// TIA Portal project "phanloai_demo" (V16)

(* hardware
DEVICE "S7-1200 station_1"  S7-1200 Station
   slot 0: "Rack_0"  S7-1200 Rack  Rack  V1.0
   slot 1: "PLC_1"  CPU 1214C DC/DC/DC  6ES7 214-1AG40-0XB0  V4.4
*)

// ===== PLC "PLC_1"  CPU 1214C DC/DC/DC =====

VAR_GLOBAL   // PLC tag table "Default tag table"
   "pulse_I0.7" AT %M50.0 : Bool;
   "pulse_nanglen1" AT %M50.4 : Bool;
   "pulse_haxuong" AT %M50.5 : Bool;
   "pulse_nanglen2" AT %M50.6 : Bool;
   "pulse_haxuong1" AT %M51.0 : Bool;
   "pulse_dira" AT %M51.2 : Bool;
   "pulse_covat" AT %M61.2 : Bool;
   "pulse_vatcuoi" AT %M62.3 : Bool;
   "pulse_run" AT %M62.4 : Bool;
   "pulse_MQTT_VT2" AT %M70.1 : Bool;
   "pulse_MQTT_VT1" AT %M70.0 : Bool;
   "pulse_MQTT_VT3" AT %M70.2 : Bool;
   "pulse_VT1" AT %M63.0 : Bool;
   "pulse_dive" AT %M62.5 : Bool;
   "Tag_3" AT %M51.4 : Bool;
   "pulse_VT2" AT %M63.1 : Bool;
   "pulse_VT3" AT %M63.2 : Bool;
   "pulse_nanglen_2" AT %M62.6 : Bool;
   "Tag_5" AT %M62.7 : Bool;
   "pulse_emer" AT %M9.3 : Bool;
   "Tag_4" AT %M9.4 : Bool;
   "Tag_6" AT %M15.0 : Bool;
   "Tag_7" AT %M15.1 : Bool;
   "Tag_8" AT %M15.2 : Bool;
   "undefine" AT %M2.5 : Bool;
   "Tag_9" AT %M2.6 : Bool;
   "Tag_10" AT %M2.7 : Bool;
   "ready" AT %M4.7 : Bool;
   "not_ready" AT %M4.6 : Bool;
   "Tag_11" AT %M5.5 : Bool;
   "Tag_12" AT %M5.6 : Bool;
   "Tag_13" AT %M5.7 : Bool;
   "stop_QR" AT %M9.5 : Bool;
   "QR_check" AT %M9.6 : Bool;
   "mode" AT %M9.7 : Bool;
   "Color_check" AT %M12.5 : Bool;
END_VAR

VAR_GLOBAL   // PLC tag table "Input"
   "Button_start" AT %I0.0 : Bool;
   "CB_covat" AT %I0.1 : Bool;
   "CB_dua_vat_ve" AT %I0.2 : Bool;
   "CB_day_vat_ra" AT %I0.3 : Bool;
   "CB_dira_2" AT %I0.4 : Bool;
   "CB_vatcuoi" AT %I0.7 : Bool;
   "CB_dive" AT %I1.0 : Bool;
   "CB_dira_1" AT %I1.1 : Bool;
   "CB_dira_3" AT %I1.2 : Bool;
   "CB_nanglen" AT %I1.3 : Bool;
   "CB_haxuong" AT %I1.4 : Bool;
   "Button_reset" AT %I1.5 : Bool;
END_VAR

VAR_GLOBAL   // PLC tag table "Output"
   "motor" AT %Q0.0 : Bool;
   "kep_phoi" AT %Q0.1 : Bool;
   "nanglen" AT %Q0.2 : Bool;
   "dive" AT %Q0.3 : Bool;
   "day_vat_ra" AT %Q0.4 : Bool;
   "nha_phoi" AT %Q0.5 : Bool;
   "haxuong" AT %Q0.6 : Bool;
   "dira" AT %Q0.7 : Bool;
   "dua_vat_ve" AT %Q1.1 : Bool;
END_VAR

VAR_GLOBAL   // PLC tag table "Memory"
   "Tag_1" AT %M0.0 : Bool;
   "Tag_2" AT %M0.1 : Bool;
   "reset_run" AT %M1.0 : Bool;
   "M_day_vat_ve" AT %M1.1 : Bool;
   "M_day_vat_ra" AT %M1.4 : Bool;
   "ha_xuong_1" AT %M2.0 : Bool;
   "nang_len_1" AT %M2.1 : Bool;
   "ha_xuong_2" AT %M2.2 : Bool;
   "nang_len_2" AT %M2.3 : Bool;
   "M_dive" AT %M2.4 : Bool;
   "dua_vat_ve_reset" AT %M3.0 : Bool;
   "nang_len_reset" AT %M3.1 : Bool;
   "dive_reset" AT %M3.2 : Bool;
   "nha_phoi_reset" AT %M3.3 : Bool;
   "co_vat" AT %M3.4 : Bool;
   "Run" AT %M3.5 : Bool;
   "motor_on" AT %M10.0 : Bool;
   "dayvat_ra_on" AT %M10.1 : Bool;
   "duavat_ve_on" AT %M10.2 : Bool;
   "dive_on" AT %M10.3 : Bool;
   "dira_on" AT %M10.4 : Bool;
   "nanglen_on" AT %M10.5 : Bool;
   "haxuong_on" AT %M10.6 : Bool;
   "kep_phoi_on" AT %M10.7 : Bool;
   "nha_phoi_on" AT %M11.0 : Bool;
   "SP1" AT %M12.0 : Bool;
   "dira_stop" AT %M12.1 : Bool;
   "VT1" AT %M12.2 : Bool;
   "VT2" AT %M12.3 : Bool;
   "VT3" AT %M12.4 : Bool;
   "M_stop" AT %M1.2 : Bool;
   "SL_VT1" AT %MW150 : UInt;
   "SL_VT2" AT %MW152 : UInt;
   "SL_VT3" AT %MW154 : UInt;
   "off_nha_phoi" AT %M3.6 : Bool;
   "off_nang_len" AT %M3.7 : Bool;
   "Auto_mode" AT %M1.3 : Bool;
   "Man_mode" AT %M1.7 : Bool;
   "Auto_run" AT %M4.0 : Bool;
   "Man_run" AT %M4.1 : Bool;
   "reset_VT1" AT %M4.2 : Bool;
   "reset_VT2" AT %M4.3 : Bool;
   "reset_VT3" AT %M4.4 : Bool;
   "stop_reset" AT %M4.5 : Bool;
   "Emer_on" AT %M5.0 : Bool;
   "Emer_run" AT %M5.2 : Bool;
   "Emer_off" AT %M5.1 : Bool;
   "S1" AT %M8.0 : Bool;
   "S2" AT %M8.1 : Bool;
   "S3" AT %M8.2 : Bool;
   "S5" AT %M8.4 : Bool;
   "S4" AT %M8.3 : Bool;
   "S6" AT %M8.5 : Bool;
   "S10" AT %M9.1 : Bool;
   "S9" AT %M9.0 : Bool;
   "S8" AT %M8.7 : Bool;
   "S7" AT %M8.6 : Bool;
END_VAR

DATA_BLOCK "Receive data MQTT"   // DB1
{ S7_Optimized_Access := 'FALSE' }
VERSION : 0.1
   VAR
      VT1 : Bool;
      VT2 : Bool;
      VT3 : Bool;
      Start : Bool;
      Stop : Bool;
      Reset : Bool;
      Emergency : Bool;
      Man_day_vat_ra : Bool;
      Man_dua_vat_ve : Bool;
      Man_haxuong : Bool;
      Man_nanglen : Bool;
      Man_kepphoi : Bool;
      Man_nhaphoi : Bool;
      Man_dira : Bool;
      Man_dive : Bool;
      Man_bangtai : Bool;
   END_VAR
BEGIN
END_DATA_BLOCK

DATA_BLOCK "Send data MQTT"   // DB2
{ S7_Optimized_Access := 'FALSE' }
VERSION : 0.1
   VAR
      SL_VT1 : Int;
      SL_VT2 : Int;
      SL_VT3 : Int;
   END_VAR
BEGIN
END_DATA_BLOCK

DATA_BLOCK "Manual"   // DB4
{ S7_Optimized_Access := 'FALSE' }
VERSION : 0.1
   VAR
      Man_motor_on : Bool;
      Man_motor_off : Bool;
      Man_dua_vat_ve : Bool;
      Man_day_vat_ra : Bool;
      Man_haxuong : Bool;
      Man_nanglen : Bool;
      Man_kepphoi : Bool;
      Man_nhaphoi : Bool;
      Man_dira : Bool;
      Man_dive : Bool;
   END_VAR
BEGIN
END_DATA_BLOCK

// folder: System blocks/Program resources

DATA_BLOCK "QR_delay"   // DB3
{ S7_Optimized_Access := 'TRUE' }
AUTHOR : Simatic
FAMILY : IEC
NAME : IEC_TMR
VERSION : 1.0
// stored: InstanceOfName IEC_TIMER
"IEC_TIMER"
BEGIN
END_DATA_BLOCK

DATA_BLOCK "QR_stop"   // DB5
{ S7_Optimized_Access := 'TRUE' }
AUTHOR : Simatic
FAMILY : IEC
NAME : IEC_TMR
VERSION : 1.0
// stored: InstanceOfName IEC_TIMER
"IEC_TIMER"
BEGIN
END_DATA_BLOCK

// folder: (top level)

FUNCTION "Auto" : Void   // FC1, LAD
{ S7_Optimized_Access := 'TRUE' }
VERSION : 0.1
   VAR_INPUT
      Button_start : Bool;
      CB_covat : Bool;
      CB_dua_vat_ve : Bool;
      CB_day_vat_ra : Bool;
      CB_dira_2 : Bool;
      CB_vatcuoi : Bool;
      CB_dive : Bool;
      CB_dira_1 : Bool;
      CB_dira_3 : Bool;
      CB_nanglen : Bool;
      CB_haxuong : Bool;
      MQTT_VT1 : Bool;
      MQTT_VT2 : Bool;
      MQTT_VT3 : Bool;
      MQTT_start : Bool;
      MQTT_stop : Bool;
      MQTT_emer : Bool;
      reset_run : Bool;
      Emer_on : Bool;
      Emer_run : Bool;
   END_VAR
   VAR_OUTPUT
      motor : Bool;
      nanglen : Bool;
      haxuong : Bool;
   END_VAR
   VAR_IN_OUT
      SL_VT1 : Int;
      SL_VT2 : Int;
      SL_VT3 : Int;
      day_vat_ra : Bool;
      dua_vat_ve : Bool;
      kep_phoi : Bool;
      dira : Bool;
      nha_phoi : Bool;
      dive : Bool;
   END_VAR
   VAR_TEMP   // added for the SCL form of the ladder/FBD networks
      _w1 : Bool;
      _w2 : Bool;
      _w3 : Bool;
      _w4 : Bool;
      _w5 : Bool;
   END_VAR
BEGIN

REGION Network 1
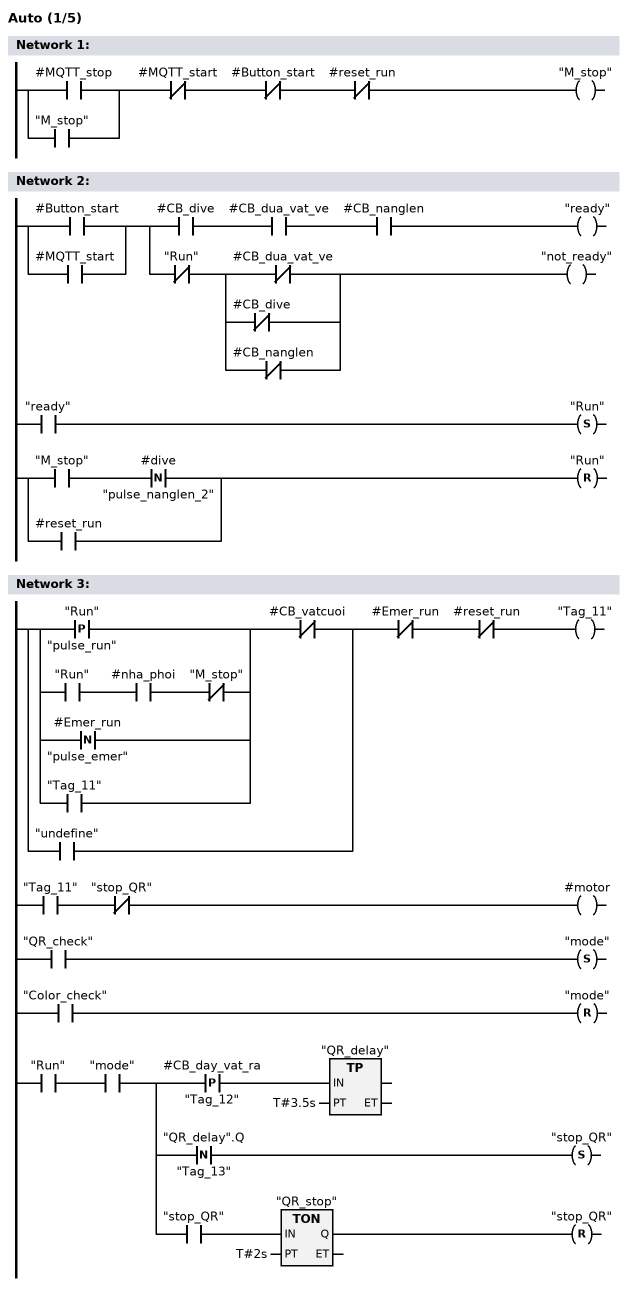
   RUNG wire#powerrail
      Contact( #MQTT_stop )
      wire#w1
      I_Contact( #MQTT_start )
      I_Contact( #Button_start )
      I_Contact( #reset_run )
      Coil( "M_stop" )
   END_RUNG
   RUNG wire#powerrail
      Contact( "M_stop" )
   END_RUNG wire#w1
   // the same network as SCL:
   "M_stop" := (#MQTT_stop OR "M_stop") AND NOT #MQTT_start AND NOT #Button_start AND NOT #reset_run;
END_REGION

REGION Network 2
   RUNG wire#powerrail
      Contact( #Button_start )
      wire#w1
      Contact( #CB_dive )
      Contact( #CB_dua_vat_ve )
      Contact( #CB_nanglen )
      Coil( "ready" )
   END_RUNG
   RUNG wire#powerrail
      Contact( #MQTT_start )
   END_RUNG wire#w1
   RUNG wire#w1
      I_Contact( "Run" )
      wire#w2
      I_Contact( #CB_dua_vat_ve )
      wire#w3
      Coil( "not_ready" )
   END_RUNG
   RUNG wire#w2
      I_Contact( #CB_dive )
   END_RUNG wire#w3
   RUNG wire#w2
      I_Contact( #CB_nanglen )
   END_RUNG wire#w3
   RUNG wire#powerrail
      Contact( "ready" )
      S_Coil( "Run" )
   END_RUNG
   RUNG wire#powerrail
      Contact( "M_stop" )
      N_Contact(operand := #dive, bit := "pulse_nanglen_2")
      wire#w4
      R_Coil( "Run" )
   END_RUNG
   RUNG wire#powerrail
      Contact( #reset_run )
   END_RUNG wire#w4
   // the same network as SCL:
   #_w1 := #Button_start OR #MQTT_start;
   "ready" := #_w1 AND #CB_dive AND #CB_dua_vat_ve AND #CB_nanglen;
   "not_ready" := #_w1 AND NOT "Run" AND (NOT #CB_dua_vat_ve OR NOT #CB_dive OR NOT #CB_nanglen);
   IF "ready" THEN "Run" := TRUE; END_IF;
   #_w2 := "M_stop" AND NOT #dive AND "pulse_nanglen_2";   // falling edge of #dive
   "pulse_nanglen_2" := #dive;
   IF #_w2 OR #reset_run THEN "Run" := FALSE; END_IF;
END_REGION

REGION Network 3
   #_w1 := "Run" AND NOT "pulse_run";   // rising edge of "Run"
   "pulse_run" := "Run";
   #_w2 := NOT #Emer_run AND "pulse_emer";   // falling edge of #Emer_run
   "pulse_emer" := #Emer_run;
   "Tag_11" := (((#_w1 OR ("Run" AND #nha_phoi AND NOT "M_stop") OR #_w2 OR "Tag_11") AND NOT #CB_vatcuoi) OR "undefine") AND NOT #Emer_run AND NOT #reset_run;
   #motor := "Tag_11" AND NOT "stop_QR";
   IF "QR_check" THEN "mode" := TRUE; END_IF;
   IF "Color_check" THEN "mode" := FALSE; END_IF;
   #_w3 := "Run" AND "mode";
   #_w4 := #_w3 AND #CB_day_vat_ra AND NOT "Tag_12";   // rising edge of #CB_day_vat_ra
   "Tag_12" := #CB_day_vat_ra;
   "QR_delay".TP(IN := #_w4, PT := T#3.5s);
   #_w5 := #_w3 AND NOT "QR_delay".Q AND "Tag_13";   // falling edge of "QR_delay".Q
   "Tag_13" := "QR_delay".Q;
   IF #_w5 THEN "stop_QR" := TRUE; END_IF;
   "QR_stop".TON(IN := #_w3 AND "stop_QR", PT := T#2s);
   IF "QR_stop".Q THEN "stop_QR" := FALSE; END_IF;
END_REGION

REGION Network 4
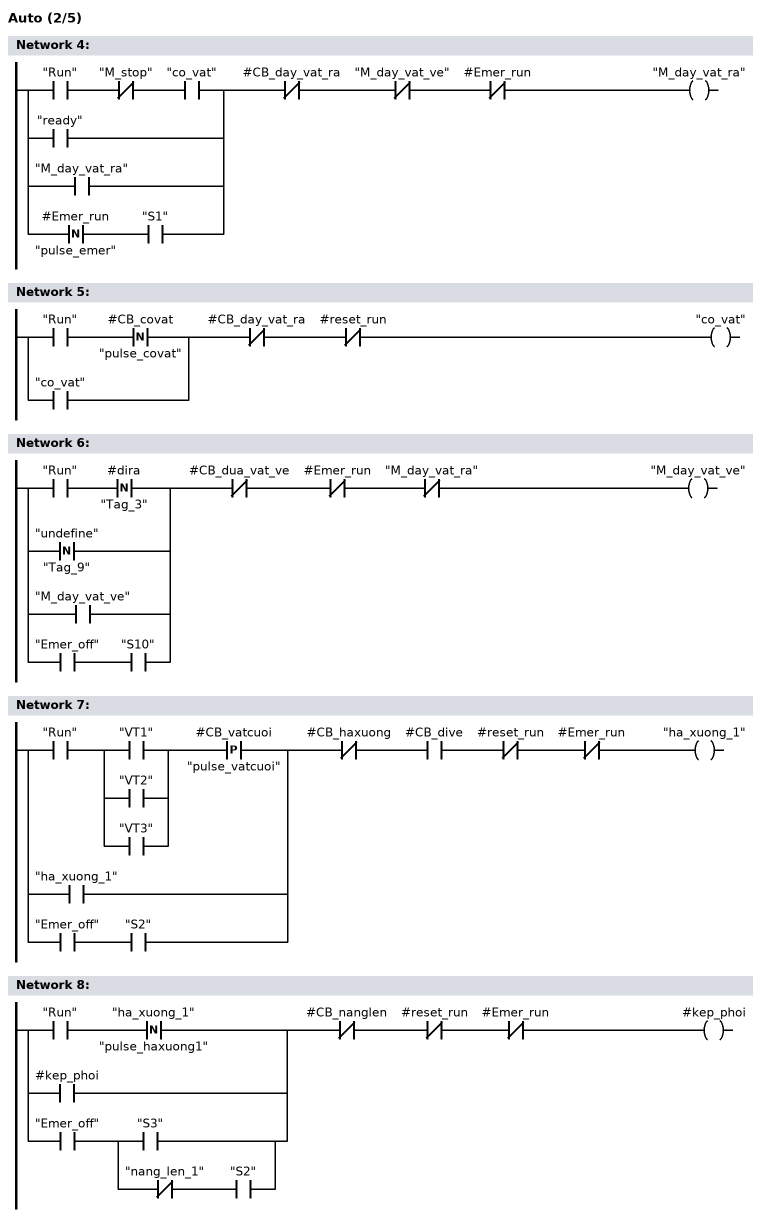
   RUNG wire#powerrail
      Contact( "Run" )
      I_Contact( "M_stop" )
      Contact( "co_vat" )
      wire#w1
      I_Contact( #CB_day_vat_ra )
      I_Contact( "M_day_vat_ve" )
      I_Contact( #Emer_run )
      Coil( "M_day_vat_ra" )
   END_RUNG
   RUNG wire#powerrail
      Contact( "ready" )
   END_RUNG wire#w1
   RUNG wire#powerrail
      Contact( "M_day_vat_ra" )
   END_RUNG wire#w1
   RUNG wire#powerrail
      N_Contact(operand := #Emer_run, bit := "pulse_emer")
      Contact( "S1" )
   END_RUNG wire#w1
   // the same network as SCL:
   #_w1 := NOT #Emer_run AND "pulse_emer";   // falling edge of #Emer_run
   "pulse_emer" := #Emer_run;
   "M_day_vat_ra" := (("Run" AND NOT "M_stop" AND "co_vat") OR "ready" OR "M_day_vat_ra" OR (#_w1 AND "S1")) AND NOT #CB_day_vat_ra AND NOT "M_day_vat_ve" AND NOT #Emer_run;
END_REGION

REGION Network 5
   RUNG wire#powerrail
      Contact( "Run" )
      N_Contact(operand := #CB_covat, bit := "pulse_covat")
      wire#w1
      I_Contact( #CB_day_vat_ra )
      I_Contact( #reset_run )
      Coil( "co_vat" )
   END_RUNG
   RUNG wire#powerrail
      Contact( "co_vat" )
   END_RUNG wire#w1
   // the same network as SCL:
   #_w1 := "Run" AND NOT #CB_covat AND "pulse_covat";   // falling edge of #CB_covat
   "pulse_covat" := #CB_covat;
   "co_vat" := (#_w1 OR "co_vat") AND NOT #CB_day_vat_ra AND NOT #reset_run;
END_REGION

REGION Network 6
   RUNG wire#powerrail
      Contact( "Run" )
      N_Contact(operand := #dira, bit := "Tag_3")
      wire#w1
      I_Contact( #CB_dua_vat_ve )
      I_Contact( #Emer_run )
      I_Contact( "M_day_vat_ra" )
      Coil( "M_day_vat_ve" )
   END_RUNG
   RUNG wire#powerrail
      N_Contact(operand := "undefine", bit := "Tag_9")
   END_RUNG wire#w1
   RUNG wire#powerrail
      Contact( "M_day_vat_ve" )
   END_RUNG wire#w1
   RUNG wire#powerrail
      Contact( "Emer_off" )
      Contact( "S10" )
   END_RUNG wire#w1
   // the same network as SCL:
   #_w1 := "Run" AND NOT #dira AND "Tag_3";   // falling edge of #dira
   "Tag_3" := #dira;
   #_w2 := NOT "undefine" AND "Tag_9";   // falling edge of "undefine"
   "Tag_9" := "undefine";
   "M_day_vat_ve" := (#_w1 OR #_w2 OR "M_day_vat_ve" OR ("Emer_off" AND "S10")) AND NOT #CB_dua_vat_ve AND NOT #Emer_run AND NOT "M_day_vat_ra";
END_REGION

REGION Network 7
   RUNG wire#powerrail
      Contact( "Run" )
      wire#w1
      Contact( "VT1" )
      wire#w2
      P_Contact(operand := #CB_vatcuoi, bit := "pulse_vatcuoi")
      wire#w3
      I_Contact( #CB_haxuong )
      Contact( #CB_dive )
      I_Contact( #reset_run )
      I_Contact( #Emer_run )
      Coil( "ha_xuong_1" )
   END_RUNG
   RUNG wire#w1
      Contact( "VT2" )
   END_RUNG wire#w2
   RUNG wire#w1
      Contact( "VT3" )
   END_RUNG wire#w2
   RUNG wire#powerrail
      Contact( "ha_xuong_1" )
   END_RUNG wire#w3
   RUNG wire#powerrail
      Contact( "Emer_off" )
      Contact( "S2" )
   END_RUNG wire#w3
   // the same network as SCL:
   #_w1 := "Run" AND ("VT1" OR "VT2" OR "VT3") AND #CB_vatcuoi AND NOT "pulse_vatcuoi";   // rising edge of #CB_vatcuoi
   "pulse_vatcuoi" := #CB_vatcuoi;
   "ha_xuong_1" := (#_w1 OR "ha_xuong_1" OR ("Emer_off" AND "S2")) AND NOT #CB_haxuong AND #CB_dive AND NOT #reset_run AND NOT #Emer_run;
END_REGION

REGION Network 8
   RUNG wire#powerrail
      Contact( "Run" )
      N_Contact(operand := "ha_xuong_1", bit := "pulse_haxuong1")
      wire#w1
      I_Contact( #CB_nanglen )
      I_Contact( #reset_run )
      I_Contact( #Emer_run )
      Coil( #kep_phoi )
   END_RUNG
   RUNG wire#powerrail
      Contact( #kep_phoi )
   END_RUNG wire#w1
   RUNG wire#powerrail
      Contact( "Emer_off" )
      wire#w2
      Contact( "S3" )
   END_RUNG wire#w1
   RUNG wire#w2
      I_Contact( "nang_len_1" )
      Contact( "S2" )
   END_RUNG wire#w1
   // the same network as SCL:
   #_w1 := "Run" AND NOT "ha_xuong_1" AND "pulse_haxuong1";   // falling edge of "ha_xuong_1"
   "pulse_haxuong1" := "ha_xuong_1";
   #kep_phoi := (#_w1 OR #kep_phoi OR ("Emer_off" AND ("S3" OR (NOT "nang_len_1" AND "S2")))) AND NOT #CB_nanglen AND NOT #reset_run AND NOT #Emer_run;
END_REGION

REGION Network 9
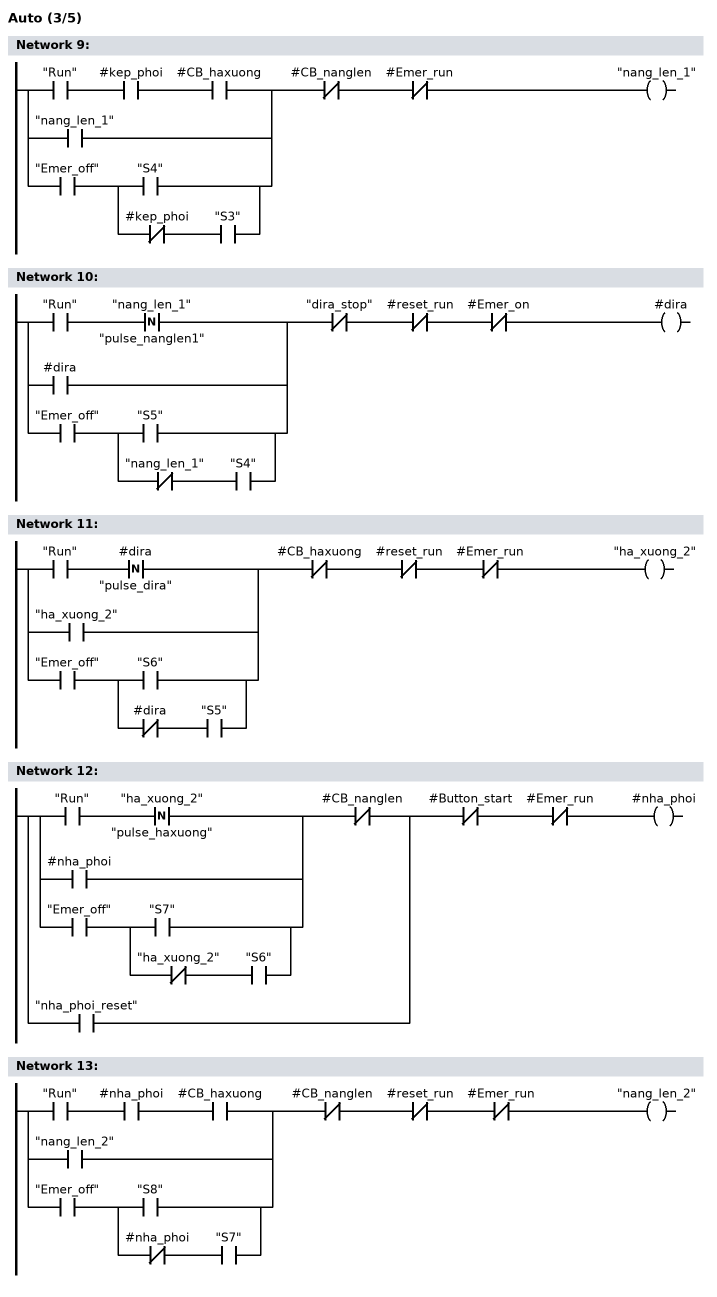
   RUNG wire#powerrail
      Contact( "Run" )
      Contact( #kep_phoi )
      Contact( #CB_haxuong )
      wire#w1
      I_Contact( #CB_nanglen )
      I_Contact( #Emer_run )
      Coil( "nang_len_1" )
   END_RUNG
   RUNG wire#powerrail
      Contact( "nang_len_1" )
   END_RUNG wire#w1
   RUNG wire#powerrail
      Contact( "Emer_off" )
      wire#w2
      Contact( "S4" )
   END_RUNG wire#w1
   RUNG wire#w2
      I_Contact( #kep_phoi )
      Contact( "S3" )
   END_RUNG wire#w1
   // the same network as SCL:
   "nang_len_1" := (("Run" AND #kep_phoi AND #CB_haxuong) OR "nang_len_1" OR ("Emer_off" AND ("S4" OR (NOT #kep_phoi AND "S3")))) AND NOT #CB_nanglen AND NOT #Emer_run;
END_REGION

REGION Network 10
   RUNG wire#powerrail
      Contact( "Run" )
      N_Contact(operand := "nang_len_1", bit := "pulse_nanglen1")
      wire#w1
      I_Contact( "dira_stop" )
      I_Contact( #reset_run )
      I_Contact( #Emer_on )
      Coil( #dira )
   END_RUNG
   RUNG wire#powerrail
      Contact( #dira )
   END_RUNG wire#w1
   RUNG wire#powerrail
      Contact( "Emer_off" )
      wire#w2
      Contact( "S5" )
   END_RUNG wire#w1
   RUNG wire#w2
      I_Contact( "nang_len_1" )
      Contact( "S4" )
   END_RUNG wire#w1
   // the same network as SCL:
   #_w1 := "Run" AND NOT "nang_len_1" AND "pulse_nanglen1";   // falling edge of "nang_len_1"
   "pulse_nanglen1" := "nang_len_1";
   #dira := (#_w1 OR #dira OR ("Emer_off" AND ("S5" OR (NOT "nang_len_1" AND "S4")))) AND NOT "dira_stop" AND NOT #reset_run AND NOT #Emer_on;
END_REGION

REGION Network 11
   RUNG wire#powerrail
      Contact( "Run" )
      N_Contact(operand := #dira, bit := "pulse_dira")
      wire#w1
      I_Contact( #CB_haxuong )
      I_Contact( #reset_run )
      I_Contact( #Emer_run )
      Coil( "ha_xuong_2" )
   END_RUNG
   RUNG wire#powerrail
      Contact( "ha_xuong_2" )
   END_RUNG wire#w1
   RUNG wire#powerrail
      Contact( "Emer_off" )
      wire#w2
      Contact( "S6" )
   END_RUNG wire#w1
   RUNG wire#w2
      I_Contact( #dira )
      Contact( "S5" )
   END_RUNG wire#w1
   // the same network as SCL:
   #_w1 := "Run" AND NOT #dira AND "pulse_dira";   // falling edge of #dira
   "pulse_dira" := #dira;
   "ha_xuong_2" := (#_w1 OR "ha_xuong_2" OR ("Emer_off" AND ("S6" OR (NOT #dira AND "S5")))) AND NOT #CB_haxuong AND NOT #reset_run AND NOT #Emer_run;
END_REGION

REGION Network 12
   RUNG wire#powerrail
      Contact( "Run" )
      N_Contact(operand := "ha_xuong_2", bit := "pulse_haxuong")
      wire#w1
      I_Contact( #CB_nanglen )
      wire#w3
      I_Contact( #Button_start )
      I_Contact( #Emer_run )
      Coil( #nha_phoi )
   END_RUNG
   RUNG wire#powerrail
      Contact( #nha_phoi )
   END_RUNG wire#w1
   RUNG wire#powerrail
      Contact( "Emer_off" )
      wire#w2
      Contact( "S7" )
   END_RUNG wire#w1
   RUNG wire#w2
      I_Contact( "ha_xuong_2" )
      Contact( "S6" )
   END_RUNG wire#w1
   RUNG wire#powerrail
      Contact( "nha_phoi_reset" )
   END_RUNG wire#w3
   // the same network as SCL:
   #_w1 := "Run" AND NOT "ha_xuong_2" AND "pulse_haxuong";   // falling edge of "ha_xuong_2"
   "pulse_haxuong" := "ha_xuong_2";
   #nha_phoi := (((#_w1 OR #nha_phoi OR ("Emer_off" AND ("S7" OR (NOT "ha_xuong_2" AND "S6")))) AND NOT #CB_nanglen) OR "nha_phoi_reset") AND NOT #Button_start AND NOT #Emer_run;
END_REGION

REGION Network 13
   RUNG wire#powerrail
      Contact( "Run" )
      Contact( #nha_phoi )
      Contact( #CB_haxuong )
      wire#w1
      I_Contact( #CB_nanglen )
      I_Contact( #reset_run )
      I_Contact( #Emer_run )
      Coil( "nang_len_2" )
   END_RUNG
   RUNG wire#powerrail
      Contact( "nang_len_2" )
   END_RUNG wire#w1
   RUNG wire#powerrail
      Contact( "Emer_off" )
      wire#w2
      Contact( "S8" )
   END_RUNG wire#w1
   RUNG wire#w2
      I_Contact( #nha_phoi )
      Contact( "S7" )
   END_RUNG wire#w1
   // the same network as SCL:
   "nang_len_2" := (("Run" AND #nha_phoi AND #CB_haxuong) OR "nang_len_2" OR ("Emer_off" AND ("S8" OR (NOT #nha_phoi AND "S7")))) AND NOT #CB_nanglen AND NOT #reset_run AND NOT #Emer_run;
END_REGION

REGION Network 14
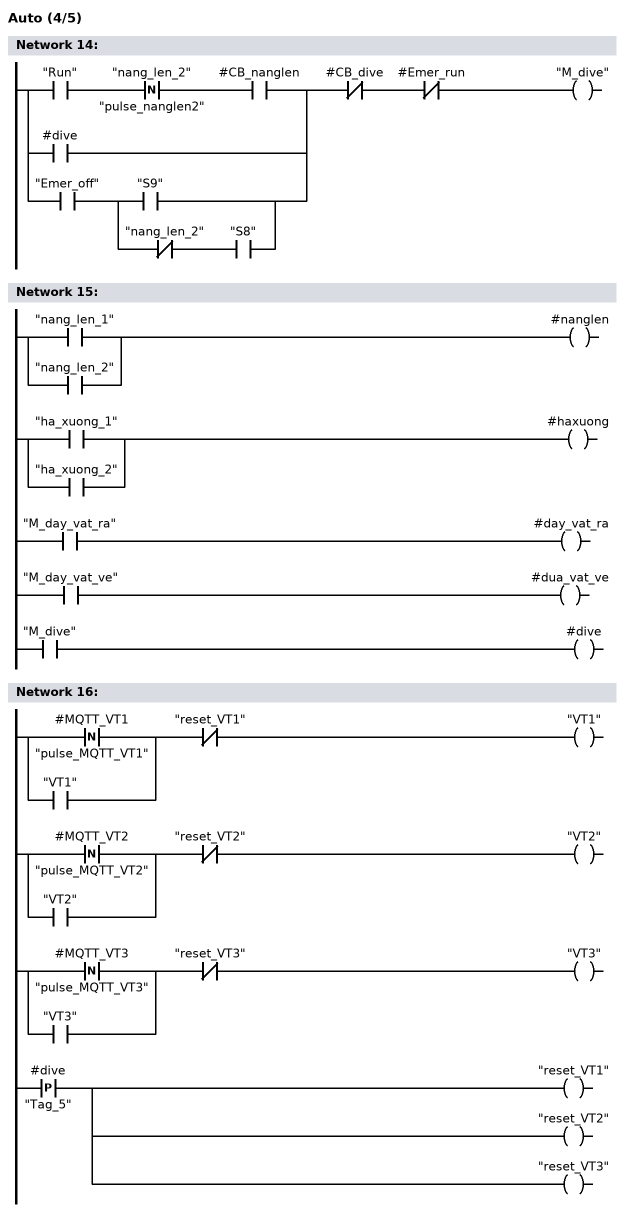
   RUNG wire#powerrail
      Contact( "Run" )
      N_Contact(operand := "nang_len_2", bit := "pulse_nanglen2")
      Contact( #CB_nanglen )
      wire#w1
      I_Contact( #CB_dive )
      I_Contact( #Emer_run )
      Coil( "M_dive" )
   END_RUNG
   RUNG wire#powerrail
      Contact( #dive )
   END_RUNG wire#w1
   RUNG wire#powerrail
      Contact( "Emer_off" )
      wire#w2
      Contact( "S9" )
   END_RUNG wire#w1
   RUNG wire#w2
      I_Contact( "nang_len_2" )
      Contact( "S8" )
   END_RUNG wire#w1
   // the same network as SCL:
   #_w1 := "Run" AND NOT "nang_len_2" AND "pulse_nanglen2";   // falling edge of "nang_len_2"
   "pulse_nanglen2" := "nang_len_2";
   "M_dive" := ((#_w1 AND #CB_nanglen) OR #dive OR ("Emer_off" AND ("S9" OR (NOT "nang_len_2" AND "S8")))) AND NOT #CB_dive AND NOT #Emer_run;
END_REGION

REGION Network 15
   RUNG wire#powerrail
      Contact( "nang_len_1" )
      wire#w1
      Coil( #nanglen )
   END_RUNG
   RUNG wire#powerrail
      Contact( "nang_len_2" )
   END_RUNG wire#w1
   RUNG wire#powerrail
      Contact( "ha_xuong_1" )
      wire#w2
      Coil( #haxuong )
   END_RUNG
   RUNG wire#powerrail
      Contact( "ha_xuong_2" )
   END_RUNG wire#w2
   RUNG wire#powerrail
      Contact( "M_day_vat_ra" )
      Coil( #day_vat_ra )
   END_RUNG
   RUNG wire#powerrail
      Contact( "M_day_vat_ve" )
      Coil( #dua_vat_ve )
   END_RUNG
   RUNG wire#powerrail
      Contact( "M_dive" )
      Coil( #dive )
   END_RUNG
   // the same network as SCL:
   #nanglen := "nang_len_1" OR "nang_len_2";
   #haxuong := "ha_xuong_1" OR "ha_xuong_2";
   #day_vat_ra := "M_day_vat_ra";
   #dua_vat_ve := "M_day_vat_ve";
   #dive := "M_dive";
END_REGION

REGION Network 16
   RUNG wire#powerrail
      N_Contact(operand := #MQTT_VT1, bit := "pulse_MQTT_VT1")
      wire#w1
      I_Contact( "reset_VT1" )
      Coil( "VT1" )
   END_RUNG
   RUNG wire#powerrail
      Contact( "VT1" )
   END_RUNG wire#w1
   RUNG wire#powerrail
      N_Contact(operand := #MQTT_VT2, bit := "pulse_MQTT_VT2")
      wire#w2
      I_Contact( "reset_VT2" )
      Coil( "VT2" )
   END_RUNG
   RUNG wire#powerrail
      Contact( "VT2" )
   END_RUNG wire#w2
   RUNG wire#powerrail
      N_Contact(operand := #MQTT_VT3, bit := "pulse_MQTT_VT3")
      wire#w3
      I_Contact( "reset_VT3" )
      Coil( "VT3" )
   END_RUNG
   RUNG wire#powerrail
      Contact( "VT3" )
   END_RUNG wire#w3
   RUNG wire#powerrail
      P_Contact(operand := #dive, bit := "Tag_5")
      wire#w4
      Coil( "reset_VT1" )
   END_RUNG
   RUNG wire#w4
      Coil( "reset_VT2" )
   END_RUNG
   RUNG wire#w4
      Coil( "reset_VT3" )
   END_RUNG
   // the same network as SCL:
   #_w1 := NOT #MQTT_VT1 AND "pulse_MQTT_VT1";   // falling edge of #MQTT_VT1
   "pulse_MQTT_VT1" := #MQTT_VT1;
   "VT1" := (#_w1 OR "VT1") AND NOT "reset_VT1";
   #_w2 := NOT #MQTT_VT2 AND "pulse_MQTT_VT2";   // falling edge of #MQTT_VT2
   "pulse_MQTT_VT2" := #MQTT_VT2;
   "VT2" := (#_w2 OR "VT2") AND NOT "reset_VT2";
   #_w3 := NOT #MQTT_VT3 AND "pulse_MQTT_VT3";   // falling edge of #MQTT_VT3
   "pulse_MQTT_VT3" := #MQTT_VT3;
   "VT3" := (#_w3 OR "VT3") AND NOT "reset_VT3";
   #_w4 := #dive AND NOT "Tag_5";   // rising edge of #dive
   "Tag_5" := #dive;
   "reset_VT1" := #_w4;
   "reset_VT2" := #_w4;
   "reset_VT3" := #_w4;
END_REGION

REGION Network 17
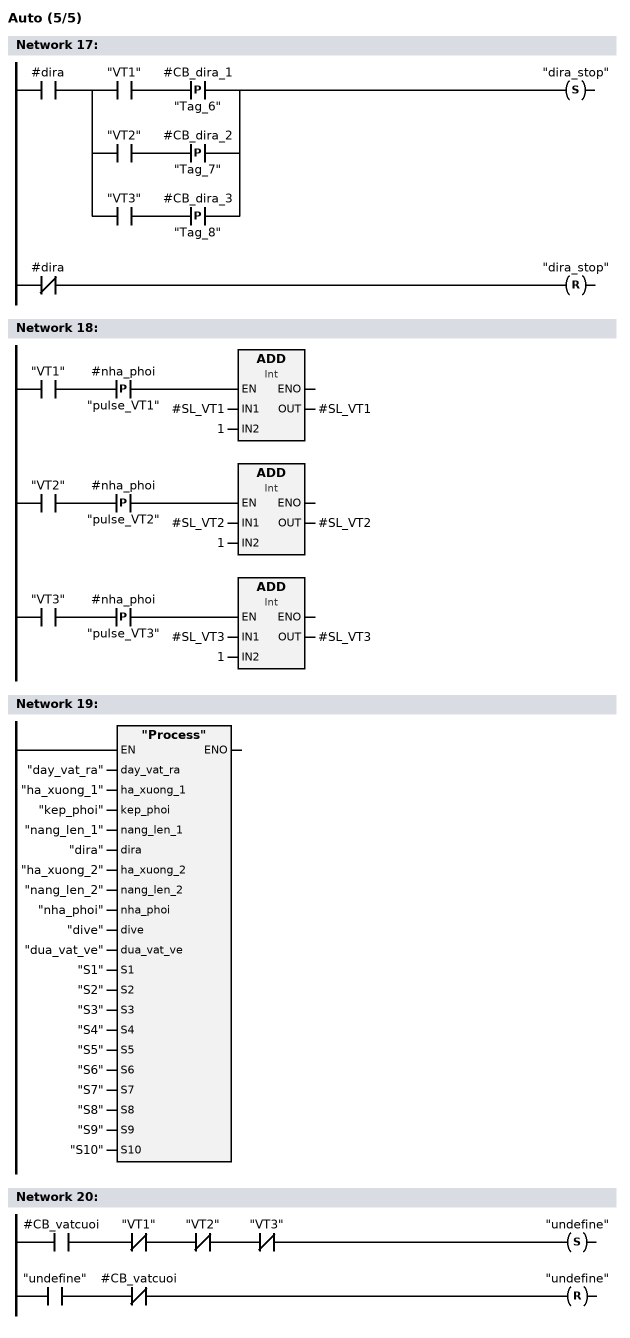
   RUNG wire#powerrail
      Contact( #dira )
      wire#w1
      Contact( "VT1" )
      P_Contact(operand := #CB_dira_1, bit := "Tag_6")
      wire#w2
      S_Coil( "dira_stop" )
   END_RUNG
   RUNG wire#w1
      Contact( "VT2" )
      P_Contact(operand := #CB_dira_2, bit := "Tag_7")
   END_RUNG wire#w2
   RUNG wire#w1
      Contact( "VT3" )
      P_Contact(operand := #CB_dira_3, bit := "Tag_8")
   END_RUNG wire#w2
   RUNG wire#powerrail
      I_Contact( #dira )
      R_Coil( "dira_stop" )
   END_RUNG
   // the same network as SCL:
   #_w1 := #dira AND "VT1" AND #CB_dira_1 AND NOT "Tag_6";   // rising edge of #CB_dira_1
   "Tag_6" := #CB_dira_1;
   #_w2 := #dira AND "VT2" AND #CB_dira_2 AND NOT "Tag_7";   // rising edge of #CB_dira_2
   "Tag_7" := #CB_dira_2;
   #_w3 := #dira AND "VT3" AND #CB_dira_3 AND NOT "Tag_8";   // rising edge of #CB_dira_3
   "Tag_8" := #CB_dira_3;
   IF #_w1 OR #_w2 OR #_w3 THEN "dira_stop" := TRUE; END_IF;
   IF NOT #dira THEN "dira_stop" := FALSE; END_IF;
END_REGION

REGION Network 18
   RUNG wire#powerrail
      Contact( "VT1" )
      P_Contact(operand := #nha_phoi, bit := "pulse_VT1")
      { S7_Templates := "SrcType := Int" } Add(in1 := #SL_VT1, in2 := 1, out => #SL_VT1)
   END_RUNG
   RUNG wire#powerrail
      Contact( "VT2" )
      P_Contact(operand := #nha_phoi, bit := "pulse_VT2")
      { S7_Templates := "SrcType := Int" } Add(in1 := #SL_VT2, in2 := 1, out => #SL_VT2)
   END_RUNG
   RUNG wire#powerrail
      Contact( "VT3" )
      P_Contact(operand := #nha_phoi, bit := "pulse_VT3")
      { S7_Templates := "SrcType := Int" } Add(in1 := #SL_VT3, in2 := 1, out => #SL_VT3)
   END_RUNG
   // the same network as SCL:
   #_w1 := "VT1" AND #nha_phoi AND NOT "pulse_VT1";   // rising edge of #nha_phoi
   "pulse_VT1" := #nha_phoi;
   IF #_w1 THEN #SL_VT1 := #SL_VT1 + 1; END_IF;
   #_w2 := "VT2" AND #nha_phoi AND NOT "pulse_VT2";   // rising edge of #nha_phoi
   "pulse_VT2" := #nha_phoi;
   IF #_w2 THEN #SL_VT2 := #SL_VT2 + 1; END_IF;
   #_w3 := "VT3" AND #nha_phoi AND NOT "pulse_VT3";   // rising edge of #nha_phoi
   "pulse_VT3" := #nha_phoi;
   IF #_w3 THEN #SL_VT3 := #SL_VT3 + 1; END_IF;
END_REGION

REGION Network 19
   RUNG wire#powerrail
      "Process"(day_vat_ra := "day_vat_ra", ha_xuong_1 := "ha_xuong_1", kep_phoi := "kep_phoi", nang_len_1 := "nang_len_1", dira := "dira", ha_xuong_2 := "ha_xuong_2", nang_len_2 := "nang_len_2", nha_phoi := "nha_phoi", dive := "dive", dua_vat_ve := "dua_vat_ve", S1 := "S1", S2 := "S2", S3 := "S3", S4 := "S4", S5 := "S5", S6 := "S6", S7 := "S7", S8 := "S8", S9 := "S9", S10 := "S10")
   END_RUNG
   // the same network as SCL:
   "Process"(day_vat_ra := "day_vat_ra",
             ha_xuong_1 := "ha_xuong_1",
             kep_phoi := "kep_phoi",
             nang_len_1 := "nang_len_1",
             dira := "dira",
             ha_xuong_2 := "ha_xuong_2",
             nang_len_2 := "nang_len_2",
             nha_phoi := "nha_phoi",
             dive := "dive",
             dua_vat_ve := "dua_vat_ve",
             S1 := "S1",
             S2 := "S2",
             S3 := "S3",
             S4 := "S4",
             S5 := "S5",
             S6 := "S6",
             S7 := "S7",
             S8 := "S8",
             S9 := "S9",
             S10 := "S10");
END_REGION

REGION Network 20
   RUNG wire#powerrail
      Contact( #CB_vatcuoi )
      I_Contact( "VT1" )
      I_Contact( "VT2" )
      I_Contact( "VT3" )
      S_Coil( "undefine" )
   END_RUNG
   RUNG wire#powerrail
      Contact( "undefine" )
      I_Contact( #CB_vatcuoi )
      R_Coil( "undefine" )
   END_RUNG
   // the same network as SCL:
   IF #CB_vatcuoi AND NOT "VT1" AND NOT "VT2" AND NOT "VT3" THEN "undefine" := TRUE; END_IF;
   IF "undefine" AND NOT #CB_vatcuoi THEN "undefine" := FALSE; END_IF;
END_REGION
END_FUNCTION

FUNCTION "Man" : Void   // FC2, LAD
{ S7_Optimized_Access := 'TRUE' }
VERSION : 0.1
   VAR_INPUT
      Man_day_vat_ra : Bool;
      Man_dua_vat_ve : Bool;
      Man_haxuong : Bool;
      Man_nanglen : Bool;
      Man_kepphoi : Bool;
      Man_nhaphoi : Bool;
      Man_dira : Bool;
      Man_dive : Bool;
      Man_motor_on : Bool;
      Man_motor_off : Bool;
      CB_covat : Bool;
      CB_dua_vat_ve : Bool;
      CB_day_vat_ra : Bool;
      CB_dira_2 : Bool;
      CB_vatcuoi : Bool;
      CB_dive : Bool;
      CB_dira_1 : Bool;
      CB_dira_3 : Bool;
      CB_nanglen : Bool;
      CB_haxuong : Bool;
      reset_run : Bool;
      emer : Bool;
   END_VAR
   VAR_IN_OUT
      dira : Bool;
      dive : Bool;
      motor : Bool;
      kep_phoi : Bool;
      nanglen : Bool;
      day_vat_ra : Bool;
      nha_phoi : Bool;
      haxuong : Bool;
      dua_vat_ve : Bool;
   END_VAR
BEGIN

REGION Network 1
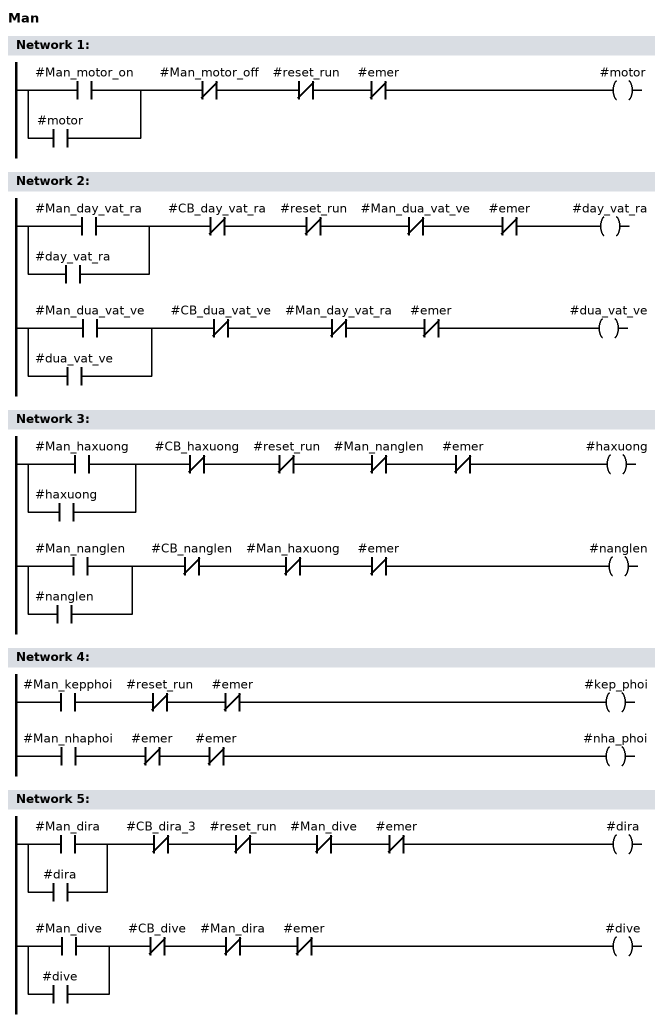
   RUNG wire#powerrail
      Contact( #Man_motor_on )
      wire#w1
      I_Contact( #Man_motor_off )
      I_Contact( #reset_run )
      I_Contact( #emer )
      Coil( #motor )
   END_RUNG
   RUNG wire#powerrail
      Contact( #motor )
   END_RUNG wire#w1
   // the same network as SCL:
   #motor := (#Man_motor_on OR #motor) AND NOT #Man_motor_off AND NOT #reset_run AND NOT #emer;
END_REGION

REGION Network 2
   RUNG wire#powerrail
      Contact( #Man_day_vat_ra )
      wire#w1
      I_Contact( #CB_day_vat_ra )
      I_Contact( #reset_run )
      I_Contact( #Man_dua_vat_ve )
      I_Contact( #emer )
      Coil( #day_vat_ra )
   END_RUNG
   RUNG wire#powerrail
      Contact( #day_vat_ra )
   END_RUNG wire#w1
   RUNG wire#powerrail
      Contact( #Man_dua_vat_ve )
      wire#w2
      I_Contact( #CB_dua_vat_ve )
      I_Contact( #Man_day_vat_ra )
      I_Contact( #emer )
      Coil( #dua_vat_ve )
   END_RUNG
   RUNG wire#powerrail
      Contact( #dua_vat_ve )
   END_RUNG wire#w2
   // the same network as SCL:
   #day_vat_ra := (#Man_day_vat_ra OR #day_vat_ra) AND NOT #CB_day_vat_ra AND NOT #reset_run AND NOT #Man_dua_vat_ve AND NOT #emer;
   #dua_vat_ve := (#Man_dua_vat_ve OR #dua_vat_ve) AND NOT #CB_dua_vat_ve AND NOT #Man_day_vat_ra AND NOT #emer;
END_REGION

REGION Network 3
   RUNG wire#powerrail
      Contact( #Man_haxuong )
      wire#w1
      I_Contact( #CB_haxuong )
      I_Contact( #reset_run )
      I_Contact( #Man_nanglen )
      I_Contact( #emer )
      Coil( #haxuong )
   END_RUNG
   RUNG wire#powerrail
      Contact( #haxuong )
   END_RUNG wire#w1
   RUNG wire#powerrail
      Contact( #Man_nanglen )
      wire#w2
      I_Contact( #CB_nanglen )
      I_Contact( #Man_haxuong )
      I_Contact( #emer )
      Coil( #nanglen )
   END_RUNG
   RUNG wire#powerrail
      Contact( #nanglen )
   END_RUNG wire#w2
   // the same network as SCL:
   #haxuong := (#Man_haxuong OR #haxuong) AND NOT #CB_haxuong AND NOT #reset_run AND NOT #Man_nanglen AND NOT #emer;
   #nanglen := (#Man_nanglen OR #nanglen) AND NOT #CB_nanglen AND NOT #Man_haxuong AND NOT #emer;
END_REGION

REGION Network 4
   RUNG wire#powerrail
      Contact( #Man_kepphoi )
      I_Contact( #reset_run )
      I_Contact( #emer )
      Coil( #kep_phoi )
   END_RUNG
   RUNG wire#powerrail
      Contact( #Man_nhaphoi )
      I_Contact( #emer )
      I_Contact( #emer )
      Coil( #nha_phoi )
   END_RUNG
   // the same network as SCL:
   #kep_phoi := #Man_kepphoi AND NOT #reset_run AND NOT #emer;
   #nha_phoi := #Man_nhaphoi AND NOT #emer AND NOT #emer;
END_REGION

REGION Network 5
   RUNG wire#powerrail
      Contact( #Man_dira )
      wire#w1
      I_Contact( #CB_dira_3 )
      I_Contact( #reset_run )
      I_Contact( #Man_dive )
      I_Contact( #emer )
      Coil( #dira )
   END_RUNG
   RUNG wire#powerrail
      Contact( #dira )
   END_RUNG wire#w1
   RUNG wire#powerrail
      Contact( #Man_dive )
      wire#w2
      I_Contact( #CB_dive )
      I_Contact( #Man_dira )
      I_Contact( #emer )
      Coil( #dive )
   END_RUNG
   RUNG wire#powerrail
      Contact( #dive )
   END_RUNG wire#w2
   // the same network as SCL:
   #dira := (#Man_dira OR #dira) AND NOT #CB_dira_3 AND NOT #reset_run AND NOT #Man_dive AND NOT #emer;
   #dive := (#Man_dive OR #dive) AND NOT #CB_dive AND NOT #Man_dira AND NOT #emer;
END_REGION
END_FUNCTION

FUNCTION "Reset" : Void   // FC3, LAD
{ S7_Optimized_Access := 'TRUE' }
VERSION : 0.1
   VAR_INPUT
      CB_dua_vat_ve : Bool;
      CB_nanglen : Bool;
      CB_dive : Bool;
      reset_run : Bool;
   END_VAR
   VAR_OUTPUT
      SL_VT1 : Int;
      SL_VT2 : Int;
      SL_VT3 : Int;
      dua_vat_ve : Bool;
      nanglen : Bool;
      dive : Bool;
      nha_phoi : Bool;
      motor : Bool;
      run : Bool;
   END_VAR
   VAR_TEMP
      off_nha_phoi : Bool;
      off_nang_len : Bool;
   END_VAR
BEGIN

REGION Network 1
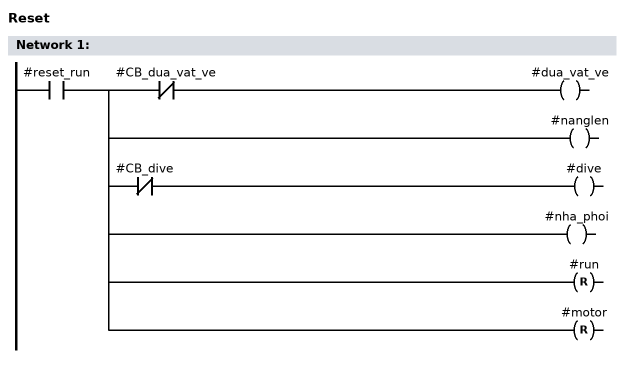
   RUNG wire#powerrail
      Contact( #reset_run )
      wire#w1
      I_Contact( #CB_dua_vat_ve )
      Coil( #dua_vat_ve )
   END_RUNG
   RUNG wire#w1
      Coil( #nanglen )
   END_RUNG
   RUNG wire#w1
      I_Contact( #CB_dive )
      Coil( #dive )
   END_RUNG
   RUNG wire#w1
      Coil( #nha_phoi )
   END_RUNG
   RUNG wire#w1
      R_Coil( #run )
   END_RUNG
   RUNG wire#w1
      R_Coil( #motor )
   END_RUNG
   // the same network as SCL:
   #dua_vat_ve := #reset_run AND NOT #CB_dua_vat_ve;
   #nanglen := #reset_run;
   #dive := #reset_run AND NOT #CB_dive;
   #nha_phoi := #reset_run;
   IF #reset_run THEN
       #run := FALSE;
       #motor := FALSE;
   END_IF;
END_REGION
END_FUNCTION

FUNCTION "Process" : Void   // FC4, LAD
{ S7_Optimized_Access := 'TRUE' }
VERSION : 0.1
   VAR_INPUT
      day_vat_ra : Bool;
      ha_xuong_1 : Bool;
      kep_phoi : Bool;
      nang_len_1 : Bool;
      dira : Bool;
      ha_xuong_2 : Bool;
      nang_len_2 : Bool;
      nha_phoi : Bool;
      dive : Bool;
      dua_vat_ve : Bool;
   END_VAR
   VAR_IN_OUT
      S1 : Bool;
      S2 : Bool;
      S3 : Bool;
      S4 : Bool;
      S5 : Bool;
      S6 : Bool;
      S7 : Bool;
      S8 : Bool;
      S9 : Bool;
      S10 : Bool;
   END_VAR
BEGIN

REGION Network 1
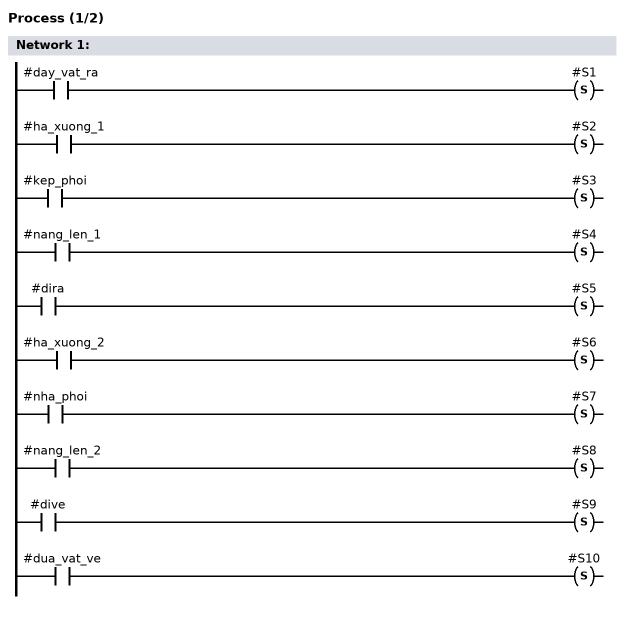
   RUNG wire#powerrail
      Contact( #day_vat_ra )
      S_Coil( #S1 )
   END_RUNG
   RUNG wire#powerrail
      Contact( #ha_xuong_1 )
      S_Coil( #S2 )
   END_RUNG
   RUNG wire#powerrail
      Contact( #kep_phoi )
      S_Coil( #S3 )
   END_RUNG
   RUNG wire#powerrail
      Contact( #nang_len_1 )
      S_Coil( #S4 )
   END_RUNG
   RUNG wire#powerrail
      Contact( #dira )
      S_Coil( #S5 )
   END_RUNG
   RUNG wire#powerrail
      Contact( #ha_xuong_2 )
      S_Coil( #S6 )
   END_RUNG
   RUNG wire#powerrail
      Contact( #nha_phoi )
      S_Coil( #S7 )
   END_RUNG
   RUNG wire#powerrail
      Contact( #nang_len_2 )
      S_Coil( #S8 )
   END_RUNG
   RUNG wire#powerrail
      Contact( #dive )
      S_Coil( #S9 )
   END_RUNG
   RUNG wire#powerrail
      Contact( #dua_vat_ve )
      S_Coil( #S10 )
   END_RUNG
   // the same network as SCL:
   IF #day_vat_ra THEN #S1 := TRUE; END_IF;
   IF #ha_xuong_1 THEN #S2 := TRUE; END_IF;
   IF #kep_phoi THEN #S3 := TRUE; END_IF;
   IF #nang_len_1 THEN #S4 := TRUE; END_IF;
   IF #dira THEN #S5 := TRUE; END_IF;
   IF #ha_xuong_2 THEN #S6 := TRUE; END_IF;
   IF #nha_phoi THEN #S7 := TRUE; END_IF;
   IF #nang_len_2 THEN #S8 := TRUE; END_IF;
   IF #dive THEN #S9 := TRUE; END_IF;
   IF #dua_vat_ve THEN #S10 := TRUE; END_IF;
END_REGION

REGION Network 2
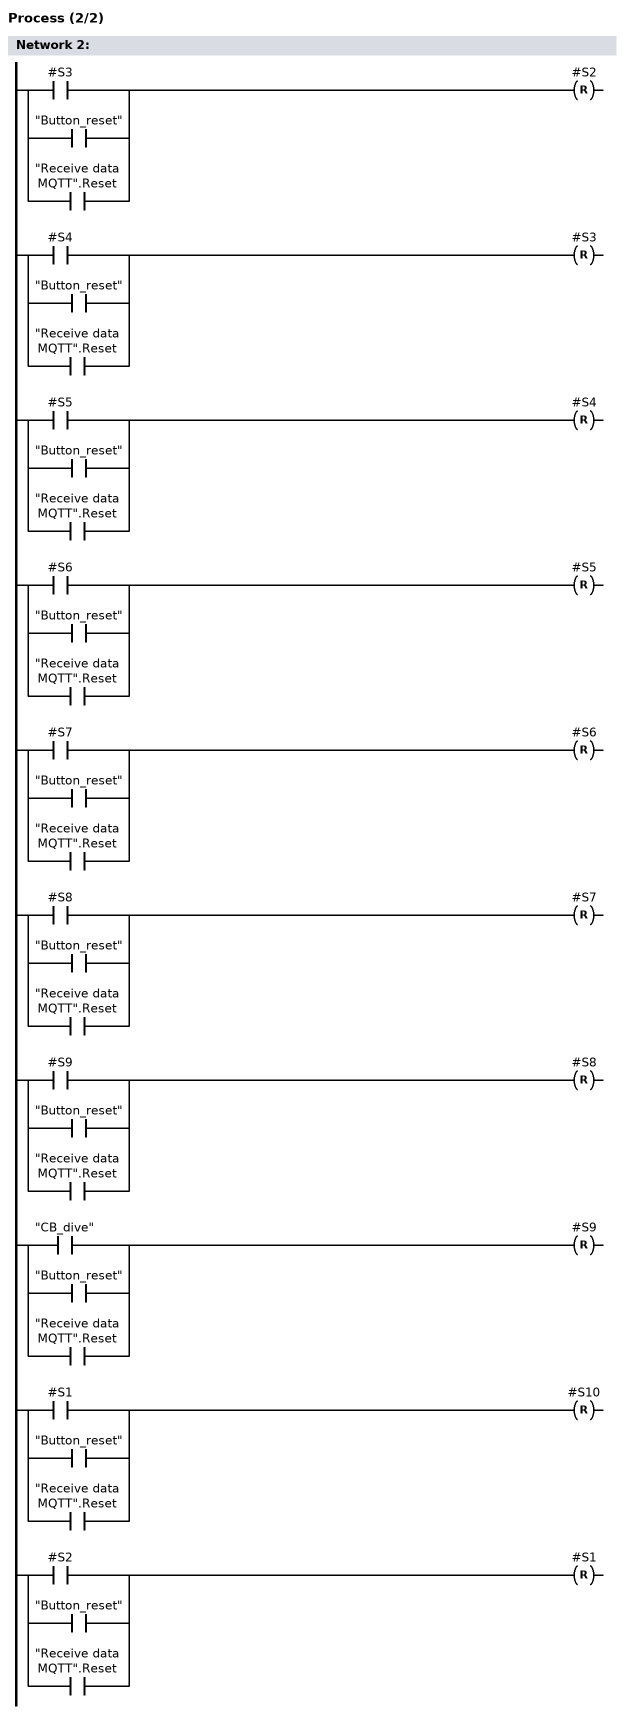
   RUNG wire#powerrail
      Contact( #S3 )
      wire#w1
      R_Coil( #S2 )
   END_RUNG
   RUNG wire#powerrail
      Contact( "Button_reset" )
   END_RUNG wire#w1
   RUNG wire#powerrail
      Contact( "Receive data MQTT".Reset )
   END_RUNG wire#w1
   RUNG wire#powerrail
      Contact( #S4 )
      wire#w2
      R_Coil( #S3 )
   END_RUNG
   RUNG wire#powerrail
      Contact( "Button_reset" )
   END_RUNG wire#w2
   RUNG wire#powerrail
      Contact( "Receive data MQTT".Reset )
   END_RUNG wire#w2
   RUNG wire#powerrail
      Contact( #S5 )
      wire#w3
      R_Coil( #S4 )
   END_RUNG
   RUNG wire#powerrail
      Contact( "Button_reset" )
   END_RUNG wire#w3
   RUNG wire#powerrail
      Contact( "Receive data MQTT".Reset )
   END_RUNG wire#w3
   RUNG wire#powerrail
      Contact( #S6 )
      wire#w4
      R_Coil( #S5 )
   END_RUNG
   RUNG wire#powerrail
      Contact( "Button_reset" )
   END_RUNG wire#w4
   RUNG wire#powerrail
      Contact( "Receive data MQTT".Reset )
   END_RUNG wire#w4
   RUNG wire#powerrail
      Contact( #S7 )
      wire#w5
      R_Coil( #S6 )
   END_RUNG
   RUNG wire#powerrail
      Contact( "Button_reset" )
   END_RUNG wire#w5
   RUNG wire#powerrail
      Contact( "Receive data MQTT".Reset )
   END_RUNG wire#w5
   RUNG wire#powerrail
      Contact( #S8 )
      wire#w6
      R_Coil( #S7 )
   END_RUNG
   RUNG wire#powerrail
      Contact( "Button_reset" )
   END_RUNG wire#w6
   RUNG wire#powerrail
      Contact( "Receive data MQTT".Reset )
   END_RUNG wire#w6
   RUNG wire#powerrail
      Contact( #S9 )
      wire#w7
      R_Coil( #S8 )
   END_RUNG
   RUNG wire#powerrail
      Contact( "Button_reset" )
   END_RUNG wire#w7
   RUNG wire#powerrail
      Contact( "Receive data MQTT".Reset )
   END_RUNG wire#w7
   RUNG wire#powerrail
      Contact( "CB_dive" )
      wire#w8
      R_Coil( #S9 )
   END_RUNG
   RUNG wire#powerrail
      Contact( "Button_reset" )
   END_RUNG wire#w8
   RUNG wire#powerrail
      Contact( "Receive data MQTT".Reset )
   END_RUNG wire#w8
   RUNG wire#powerrail
      Contact( #S1 )
      wire#w9
      R_Coil( #S10 )
   END_RUNG
   RUNG wire#powerrail
      Contact( "Button_reset" )
   END_RUNG wire#w9
   RUNG wire#powerrail
      Contact( "Receive data MQTT".Reset )
   END_RUNG wire#w9
   RUNG wire#powerrail
      Contact( #S2 )
      wire#w10
      R_Coil( #S1 )
   END_RUNG
   RUNG wire#powerrail
      Contact( "Button_reset" )
   END_RUNG wire#w10
   RUNG wire#powerrail
      Contact( "Receive data MQTT".Reset )
   END_RUNG wire#w10
   // the same network as SCL:
   IF #S3 OR "Button_reset" OR "Receive data MQTT".Reset THEN #S2 := FALSE; END_IF;
   IF #S4 OR "Button_reset" OR "Receive data MQTT".Reset THEN #S3 := FALSE; END_IF;
   IF #S5 OR "Button_reset" OR "Receive data MQTT".Reset THEN #S4 := FALSE; END_IF;
   IF #S6 OR "Button_reset" OR "Receive data MQTT".Reset THEN #S5 := FALSE; END_IF;
   IF #S7 OR "Button_reset" OR "Receive data MQTT".Reset THEN #S6 := FALSE; END_IF;
   IF #S8 OR "Button_reset" OR "Receive data MQTT".Reset THEN #S7 := FALSE; END_IF;
   IF #S9 OR "Button_reset" OR "Receive data MQTT".Reset THEN #S8 := FALSE; END_IF;
   IF "CB_dive" OR "Button_reset" OR "Receive data MQTT".Reset THEN #S9 := FALSE; END_IF;
   IF #S1 OR "Button_reset" OR "Receive data MQTT".Reset THEN #S10 := FALSE; END_IF;
   IF #S2 OR "Button_reset" OR "Receive data MQTT".Reset THEN #S1 := FALSE; END_IF;
END_REGION
END_FUNCTION

ORGANIZATION_BLOCK "Main"   // OB1, LAD, ProgramCycle
TITLE = "Main Program Sweep (Cycle)"
{ S7_Optimized_Access := 'TRUE' }
VERSION : 0.1
   VAR_INPUT
      Initial_Call : Bool;   // Initial call of this OB
      Remanence : Bool;   // =True, if remanent data are available
   END_VAR
BEGIN

REGION Network 1
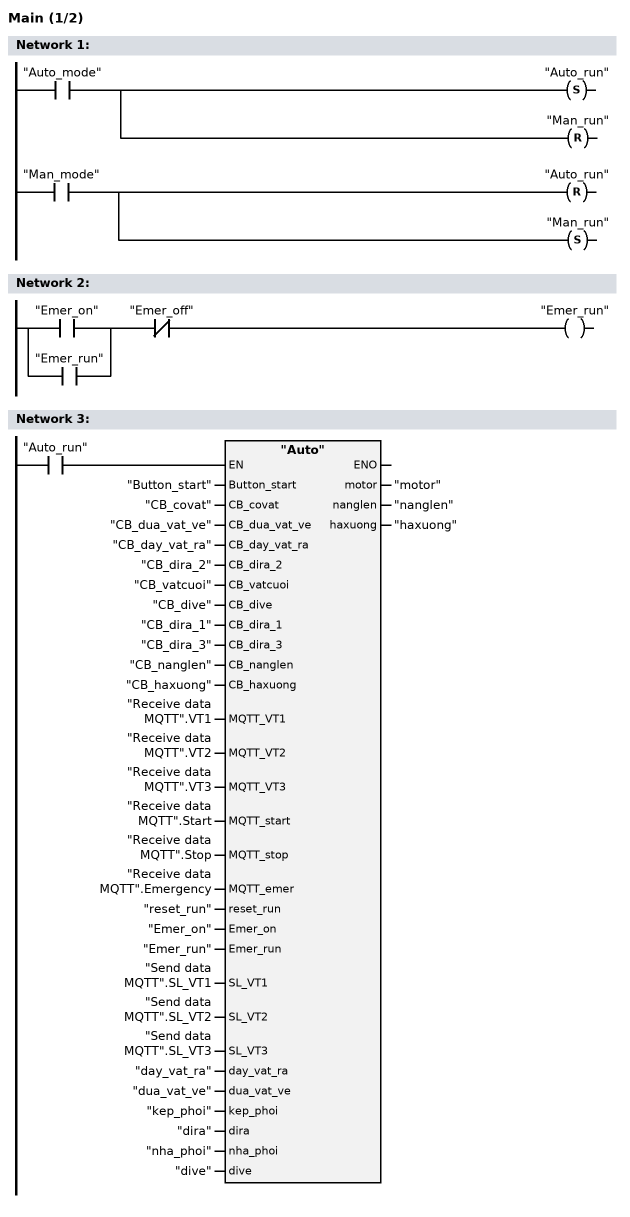
   RUNG wire#powerrail
      Contact( "Auto_mode" )
      wire#w1
      S_Coil( "Auto_run" )
   END_RUNG
   RUNG wire#w1
      R_Coil( "Man_run" )
   END_RUNG
   RUNG wire#powerrail
      Contact( "Man_mode" )
      wire#w2
      R_Coil( "Auto_run" )
   END_RUNG
   RUNG wire#w2
      S_Coil( "Man_run" )
   END_RUNG
   // the same network as SCL:
   IF "Auto_mode" THEN
       "Auto_run" := TRUE;
       "Man_run" := FALSE;
   END_IF;
   IF "Man_mode" THEN
       "Auto_run" := FALSE;
       "Man_run" := TRUE;
   END_IF;
END_REGION

REGION Network 2
   RUNG wire#powerrail
      Contact( "Emer_on" )
      wire#w1
      I_Contact( "Emer_off" )
      Coil( "Emer_run" )
   END_RUNG
   RUNG wire#powerrail
      Contact( "Emer_run" )
   END_RUNG wire#w1
   // the same network as SCL:
   "Emer_run" := ("Emer_on" OR "Emer_run") AND NOT "Emer_off";
END_REGION

REGION Network 3
   RUNG wire#powerrail
      Contact( "Auto_run" )
      "Auto"(Button_start := "Button_start", CB_covat := "CB_covat", CB_dua_vat_ve := "CB_dua_vat_ve", CB_day_vat_ra := "CB_day_vat_ra", CB_dira_2 := "CB_dira_2", CB_vatcuoi := "CB_vatcuoi", CB_dive := "CB_dive", CB_dira_1 := "CB_dira_1", CB_dira_3 := "CB_dira_3", CB_nanglen := "CB_nanglen", CB_haxuong := "CB_haxuong", MQTT_VT1 := "Receive data MQTT".VT1, MQTT_VT2 := "Receive data MQTT".VT2, MQTT_VT3 := "Receive data MQTT".VT3, MQTT_start := "Receive data MQTT".Start, MQTT_stop := "Receive data MQTT".Stop, MQTT_emer := "Receive data MQTT".Emergency, reset_run := "reset_run", Emer_on := "Emer_on", Emer_run := "Emer_run", SL_VT1 := "Send data MQTT".SL_VT1, SL_VT2 := "Send data MQTT".SL_VT2, SL_VT3 := "Send data MQTT".SL_VT3, day_vat_ra := "day_vat_ra", dua_vat_ve := "dua_vat_ve", kep_phoi := "kep_phoi", dira := "dira", nha_phoi := "nha_phoi", dive := "dive", motor => "motor", nanglen => "nanglen", haxuong => "haxuong")
   END_RUNG
   // the same network as SCL:
   IF "Auto_run" THEN
       "Auto"(Button_start := "Button_start",
              CB_covat := "CB_covat",
              CB_dua_vat_ve := "CB_dua_vat_ve",
              CB_day_vat_ra := "CB_day_vat_ra",
              CB_dira_2 := "CB_dira_2",
              CB_vatcuoi := "CB_vatcuoi",
              CB_dive := "CB_dive",
              CB_dira_1 := "CB_dira_1",
              CB_dira_3 := "CB_dira_3",
              CB_nanglen := "CB_nanglen",
              CB_haxuong := "CB_haxuong",
              MQTT_VT1 := "Receive data MQTT".VT1,
              MQTT_VT2 := "Receive data MQTT".VT2,
              MQTT_VT3 := "Receive data MQTT".VT3,
              MQTT_start := "Receive data MQTT".Start,
              MQTT_stop := "Receive data MQTT".Stop,
              MQTT_emer := "Receive data MQTT".Emergency,
              reset_run := "reset_run",
              Emer_on := "Emer_on",
              Emer_run := "Emer_run",
              SL_VT1 := "Send data MQTT".SL_VT1,
              SL_VT2 := "Send data MQTT".SL_VT2,
              SL_VT3 := "Send data MQTT".SL_VT3,
              day_vat_ra := "day_vat_ra",
              dua_vat_ve := "dua_vat_ve",
              kep_phoi := "kep_phoi",
              dira := "dira",
              nha_phoi := "nha_phoi",
              dive := "dive",
              motor => "motor",
              nanglen => "nanglen",
              haxuong => "haxuong");
   END_IF;
END_REGION

REGION Network 4
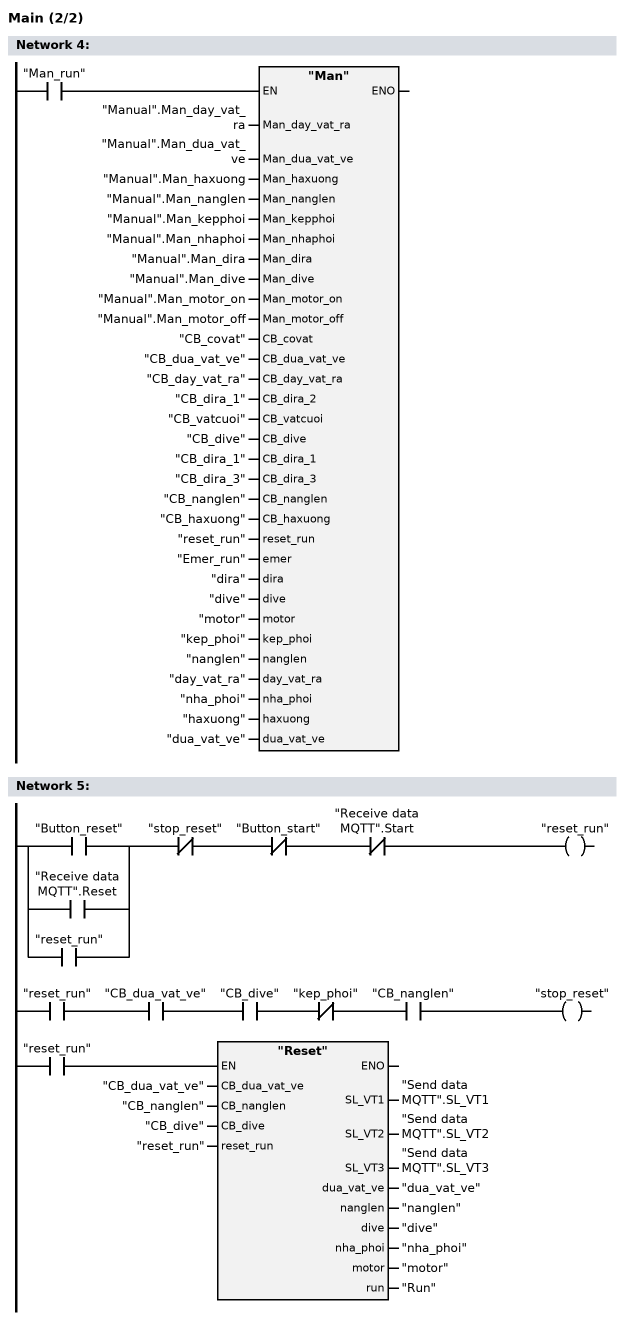
   RUNG wire#powerrail
      Contact( "Man_run" )
      "Man"(Man_day_vat_ra := "Manual".Man_day_vat_ra, Man_dua_vat_ve := "Manual".Man_dua_vat_ve, Man_haxuong := "Manual".Man_haxuong, Man_nanglen := "Manual".Man_nanglen, Man_kepphoi := "Manual".Man_kepphoi, Man_nhaphoi := "Manual".Man_nhaphoi, Man_dira := "Manual".Man_dira, Man_dive := "Manual".Man_dive, Man_motor_on := "Manual".Man_motor_on, Man_motor_off := "Manual".Man_motor_off, CB_covat := "CB_covat", CB_dua_vat_ve := "CB_dua_vat_ve", CB_day_vat_ra := "CB_day_vat_ra", CB_dira_2 := "CB_dira_1", CB_vatcuoi := "CB_vatcuoi", CB_dive := "CB_dive", CB_dira_1 := "CB_dira_1", CB_dira_3 := "CB_dira_3", CB_nanglen := "CB_nanglen", CB_haxuong := "CB_haxuong", reset_run := "reset_run", emer := "Emer_run", dira := "dira", dive := "dive", motor := "motor", kep_phoi := "kep_phoi", nanglen := "nanglen", day_vat_ra := "day_vat_ra", nha_phoi := "nha_phoi", haxuong := "haxuong", dua_vat_ve := "dua_vat_ve")
   END_RUNG
   // the same network as SCL:
   IF "Man_run" THEN
       "Man"(Man_day_vat_ra := "Manual".Man_day_vat_ra,
             Man_dua_vat_ve := "Manual".Man_dua_vat_ve,
             Man_haxuong := "Manual".Man_haxuong,
             Man_nanglen := "Manual".Man_nanglen,
             Man_kepphoi := "Manual".Man_kepphoi,
             Man_nhaphoi := "Manual".Man_nhaphoi,
             Man_dira := "Manual".Man_dira,
             Man_dive := "Manual".Man_dive,
             Man_motor_on := "Manual".Man_motor_on,
             Man_motor_off := "Manual".Man_motor_off,
             CB_covat := "CB_covat",
             CB_dua_vat_ve := "CB_dua_vat_ve",
             CB_day_vat_ra := "CB_day_vat_ra",
             CB_dira_2 := "CB_dira_1",
             CB_vatcuoi := "CB_vatcuoi",
             CB_dive := "CB_dive",
             CB_dira_1 := "CB_dira_1",
             CB_dira_3 := "CB_dira_3",
             CB_nanglen := "CB_nanglen",
             CB_haxuong := "CB_haxuong",
             reset_run := "reset_run",
             emer := "Emer_run",
             dira := "dira",
             dive := "dive",
             motor := "motor",
             kep_phoi := "kep_phoi",
             nanglen := "nanglen",
             day_vat_ra := "day_vat_ra",
             nha_phoi := "nha_phoi",
             haxuong := "haxuong",
             dua_vat_ve := "dua_vat_ve");
   END_IF;
END_REGION

REGION Network 5
   RUNG wire#powerrail
      Contact( "Button_reset" )
      wire#w1
      I_Contact( "stop_reset" )
      I_Contact( "Button_start" )
      I_Contact( "Receive data MQTT".Start )
      Coil( "reset_run" )
   END_RUNG
   RUNG wire#powerrail
      Contact( "Receive data MQTT".Reset )
   END_RUNG wire#w1
   RUNG wire#powerrail
      Contact( "reset_run" )
   END_RUNG wire#w1
   RUNG wire#powerrail
      Contact( "reset_run" )
      Contact( "CB_dua_vat_ve" )
      Contact( "CB_dive" )
      I_Contact( "kep_phoi" )
      Contact( "CB_nanglen" )
      Coil( "stop_reset" )
   END_RUNG
   RUNG wire#powerrail
      Contact( "reset_run" )
      "Reset"(CB_dua_vat_ve := "CB_dua_vat_ve", CB_nanglen := "CB_nanglen", CB_dive := "CB_dive", reset_run := "reset_run", SL_VT1 => "Send data MQTT".SL_VT1, SL_VT2 => "Send data MQTT".SL_VT2, SL_VT3 => "Send data MQTT".SL_VT3, dua_vat_ve => "dua_vat_ve", nanglen => "nanglen", dive => "dive", nha_phoi => "nha_phoi", motor => "motor", run => "Run")
   END_RUNG
   // the same network as SCL:
   "reset_run" := ("Button_reset" OR "Receive data MQTT".Reset OR "reset_run") AND NOT "stop_reset" AND NOT "Button_start" AND NOT "Receive data MQTT".Start;
   "stop_reset" := "reset_run" AND "CB_dua_vat_ve" AND "CB_dive" AND NOT "kep_phoi" AND "CB_nanglen";
   IF "reset_run" THEN
       "Reset"(CB_dua_vat_ve := "CB_dua_vat_ve",
               CB_nanglen := "CB_nanglen",
               CB_dive := "CB_dive",
               reset_run := "reset_run",
               SL_VT1 => "Send data MQTT".SL_VT1,
               SL_VT2 => "Send data MQTT".SL_VT2,
               SL_VT3 => "Send data MQTT".SL_VT3,
               dua_vat_ve => "dua_vat_ve",
               nanglen => "nanglen",
               dive => "dive",
               nha_phoi => "nha_phoi",
               motor => "motor",
               run => "Run");
   END_IF;
END_REGION
END_ORGANIZATION_BLOCK